{attribute 'GeneratedUsingTerminal: EK1122-0000-0018'}
{attribute addProperty BoxType "EK1122-0000-0018"}
{attribute addProperty Id "VI_6_AES_D_BC_ECAT_xAES_A3B0707168"}
{attribute addProperty CRC "3085977316"}
{attribute addProperty Size "68"}
{attribute addProperty Name "R7_A2_EC (EK1122)"}
TYPE R7_A2_EC_EK1122_B7F046E4 EXTENDS EK1122_1FC0878B :
STRUCT
    {attribute addProperty Name "VI-6 (AES-D-BC-ECAT)"}
    {attribute addProperty PreviousPort "R7_A2_EC (EK1122) : D"}
    {attribute addProperty SyncUnit "default"}
    VI_6_AES_D_BC_ECAT_x : AES_A3B07071;
END_STRUCT
END_TYPE

(* stored: Version 1.2.0.0, ProductVersion 3.1.4024.11
   DUT R7_A2_EC_EK1122_B7F046E4: Id {e06d499d-c881-0cc2-33d6-d6122fe744a9} *)
